// TIA Portal V17 export
// export: Created 2025-03-05T08:00:32.3052101Z, ExportSetting WithDefaults, DisplayName Totally Integrated Automation Portal, DisplayVersion V17 Update 8, DisplayName TIA Portal Openness, DisplayVersion V17 Update 8, DisplayName TIA Portal Version Control Interface, DisplayVersion V17, DisplayName SINAMICS Startdrive Advanced, DisplayVersion V17 SP2, DisplayName SINAMICS Startdrive G110M, G120, G120C, G120D, G120P, G115D, DisplayVersion V17 SP2, DisplayName SINAMICS Startdrive G130, G150, S120, S150, SINAMICS MV, S210, DisplayVersion V17 SP2, DisplayName STEP 7 Professional, DisplayVersion V17 Update 8, DisplayName SINUMERIK ONE STEP 7 Toolbox, DisplayVersion V17 Update 12, DisplayName SINUMERIK 840D sl STEP 7 Toolbox, DisplayVersion V17 Update 12, DisplayName STEP 7 Safety, DisplayVersion V17 Update 6, DisplayName WinCC Advanced, DisplayVersion V17 Update 8
FUNCTION "FC1250_UNIT_02_SEQUENCES" : Void   // FC1250, LAD
{ S7_Optimized_Access := 'FALSE' }
AUTHOR : ETXETAR
VERSION : 1.0
// stored: AutoNumber false, IsIECCheckEnabled false, SetENOAutomatically false, UDAEnableTagReadback false
BEGIN

REGION Network 1: CALL FC1253 PART CYCLE UNIT 02 CLADDING
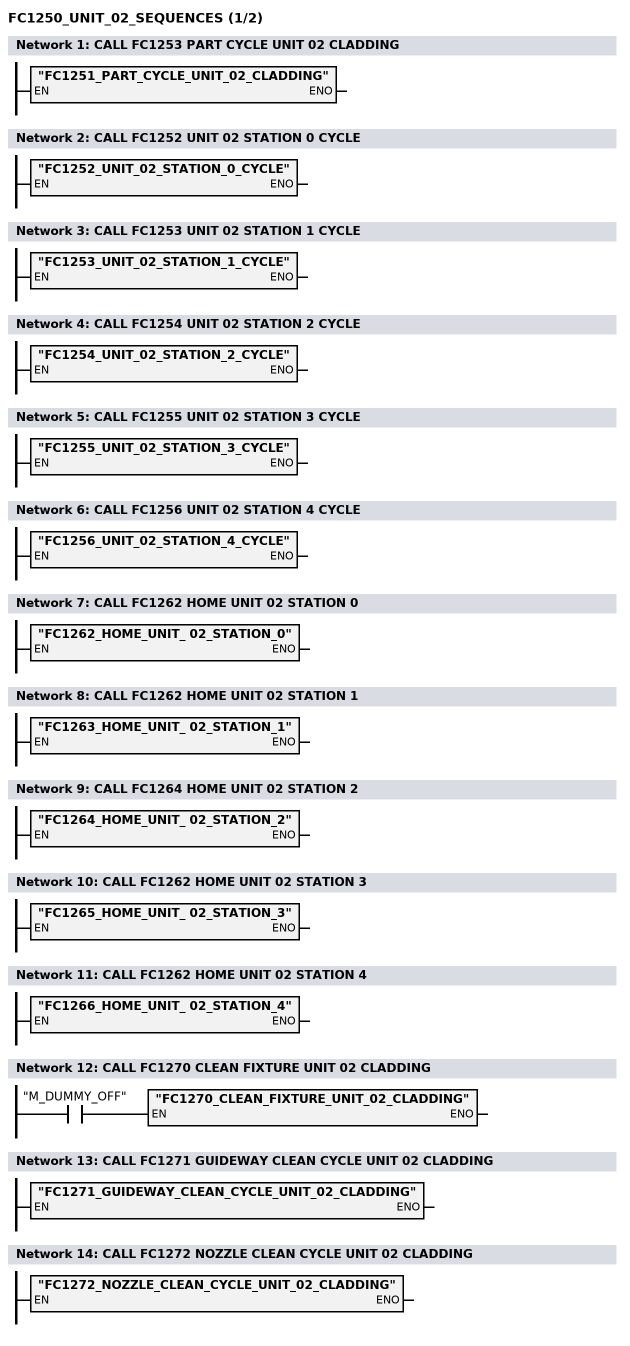
   RUNG wire#powerrail
      "FC1251_PART_CYCLE_UNIT_02_CLADDING"()
   END_RUNG
   // the same network as SCL:
   "FC1251_PART_CYCLE_UNIT_02_CLADDING"();
END_REGION

REGION Network 2: CALL FC1252 UNIT 02 STATION 0 CYCLE
   RUNG wire#powerrail
      "FC1252_UNIT_02_STATION_0_CYCLE"()
   END_RUNG
   // the same network as SCL:
   "FC1252_UNIT_02_STATION_0_CYCLE"();
END_REGION

REGION Network 3: CALL FC1253 UNIT 02 STATION 1 CYCLE
   RUNG wire#powerrail
      "FC1253_UNIT_02_STATION_1_CYCLE"()
   END_RUNG
   // the same network as SCL:
   "FC1253_UNIT_02_STATION_1_CYCLE"();
END_REGION

REGION Network 4: CALL FC1254 UNIT 02 STATION 2 CYCLE
   RUNG wire#powerrail
      "FC1254_UNIT_02_STATION_2_CYCLE"()
   END_RUNG
   // the same network as SCL:
   "FC1254_UNIT_02_STATION_2_CYCLE"();
END_REGION

REGION Network 5: CALL FC1255 UNIT 02 STATION 3 CYCLE
   RUNG wire#powerrail
      "FC1255_UNIT_02_STATION_3_CYCLE"()
   END_RUNG
   // the same network as SCL:
   "FC1255_UNIT_02_STATION_3_CYCLE"();
END_REGION

REGION Network 6: CALL FC1256 UNIT 02 STATION 4 CYCLE
   RUNG wire#powerrail
      "FC1256_UNIT_02_STATION_4_CYCLE"()
   END_RUNG
   // the same network as SCL:
   "FC1256_UNIT_02_STATION_4_CYCLE"();
END_REGION

REGION Network 7: CALL FC1262 HOME UNIT 02 STATION 0
   RUNG wire#powerrail
      "FC1262_HOME_UNIT_ 02_STATION_0"()
   END_RUNG
   // the same network as SCL:
   "FC1262_HOME_UNIT_ 02_STATION_0"();
END_REGION

REGION Network 8: CALL FC1262 HOME UNIT 02 STATION 1
   RUNG wire#powerrail
      "FC1263_HOME_UNIT_ 02_STATION_1"()
   END_RUNG
   // the same network as SCL:
   "FC1263_HOME_UNIT_ 02_STATION_1"();
END_REGION

REGION Network 9: CALL FC1264 HOME UNIT 02 STATION 2
   RUNG wire#powerrail
      "FC1264_HOME_UNIT_ 02_STATION_2"()
   END_RUNG
   // the same network as SCL:
   "FC1264_HOME_UNIT_ 02_STATION_2"();
END_REGION

REGION Network 10: CALL FC1262 HOME UNIT 02 STATION 3
   RUNG wire#powerrail
      "FC1265_HOME_UNIT_ 02_STATION_3"()
   END_RUNG
   // the same network as SCL:
   "FC1265_HOME_UNIT_ 02_STATION_3"();
END_REGION

REGION Network 11: CALL FC1262 HOME UNIT 02 STATION 4
   RUNG wire#powerrail
      "FC1266_HOME_UNIT_ 02_STATION_4"()
   END_RUNG
   // the same network as SCL:
   "FC1266_HOME_UNIT_ 02_STATION_4"();
END_REGION

REGION Network 12: CALL FC1270 CLEAN FIXTURE UNIT 02 CLADDING
   RUNG wire#powerrail
      Contact( "M_DUMMY_OFF" )
      "FC1270_CLEAN_FIXTURE_UNIT_02_CLADDING"()
   END_RUNG
   // the same network as SCL:
   IF "M_DUMMY_OFF" THEN "FC1270_CLEAN_FIXTURE_UNIT_02_CLADDING"(); END_IF;
END_REGION

REGION Network 13: CALL FC1271 GUIDEWAY CLEAN CYCLE UNIT 02 CLADDING
   RUNG wire#powerrail
      "FC1271_GUIDEWAY_CLEAN_CYCLE_UNIT_02_CLADDING"()
   END_RUNG
   // the same network as SCL:
   "FC1271_GUIDEWAY_CLEAN_CYCLE_UNIT_02_CLADDING"();
END_REGION

REGION Network 14: CALL FC1272 NOZZLE CLEAN CYCLE UNIT 02 CLADDING
   RUNG wire#powerrail
      "FC1272_NOZZLE_CLEAN_CYCLE_UNIT_02_CLADDING"()
   END_RUNG
   // the same network as SCL:
   "FC1272_NOZZLE_CLEAN_CYCLE_UNIT_02_CLADDING"();
END_REGION

REGION Network 15: CALL FC1273 MAINTENANCE UNIT 02 CLADDING
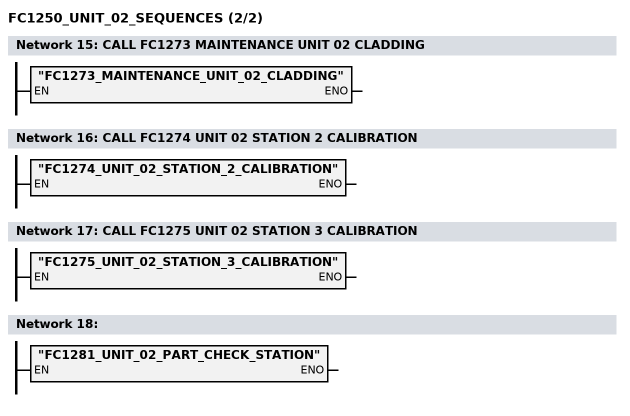
   RUNG wire#powerrail
      "FC1273_MAINTENANCE_UNIT_02_CLADDING"()
   END_RUNG
   // the same network as SCL:
   "FC1273_MAINTENANCE_UNIT_02_CLADDING"();
END_REGION

REGION Network 16: CALL FC1274 UNIT 02 STATION 2 CALIBRATION
   RUNG wire#powerrail
      "FC1274_UNIT_02_STATION_2_CALIBRATION"()
   END_RUNG
   // the same network as SCL:
   "FC1274_UNIT_02_STATION_2_CALIBRATION"();
END_REGION

REGION Network 17: CALL FC1275 UNIT 02 STATION 3 CALIBRATION
   RUNG wire#powerrail
      "FC1275_UNIT_02_STATION_3_CALIBRATION"()
   END_RUNG
   // the same network as SCL:
   "FC1275_UNIT_02_STATION_3_CALIBRATION"();
END_REGION

REGION Network 18
   RUNG wire#powerrail
      "FC1281_UNIT_02_PART_CHECK_STATION"()
   END_RUNG
   // the same network as SCL:
   "FC1281_UNIT_02_PART_CHECK_STATION"();
END_REGION
END_FUNCTION
